// TwinCAT 3 PLC project Untitled1
// ProgramVersion: 1.0.0.0
// libraries:
//   Tc2_Standard, * (Beckhoff Automation GmbH)
//   Tc2_System, * (Beckhoff Automation GmbH)
//   Tc3_GlobalTypes
//   Tc3_Module, * (Beckhoff Automation GmbH)
// project tree:
//   / PlcTask.TcTTO
//   POUs/ A_Program.TcPOU, B_Program.TcPOU, MAIN.TcPOU
// real-time tasks:
//   TASK PlcTask: cycle T#10ms, priority 20, ADS port 350

CONFIGURATION Untitled1
    RESOURCE PLC ON TwinCAT3
        TASK PlcTask(INTERVAL := T#10ms, PRIORITY := 20);
        PROGRAM MAIN WITH PlcTask : MAIN;
    END_RESOURCE
END_CONFIGURATION

// ---- POUs/MAIN.TcPOU
PROGRAM MAIN
VAR
END_VAR

A_Program();
B_Program();

END_PROGRAM

// ---- POUs/A_Program.TcPOU
PROGRAM A_Program
VAR
	i : UINT;
	x : LREAL;
	x_inc : LREAL := 0.0001;
END_VAR

FOR i := 0 TO 1000 DO
	x := x + x_inc;
END_FOR

END_PROGRAM

// ---- POUs/B_Program.TcPOU
PROGRAM B_Program
VAR
	i : UINT;
	x : LREAL;
	x_inc : LREAL := 0.0001;
	cyclecount : UINT;
END_VAR

cyclecount := cyclecount + 1;

IF cyclecount > 10 THEN
	FOR i := 0 TO 1000 DO
		x := x + x_inc;
	END_FOR	
	cyclecount := 0;
END_IF

END_PROGRAM
